# EPICS substitutions: blenApp/Db/lcls2/blen_gap_coefI2.substitutions
#======================================
# Register with DoubleVal interfaces
#======================================

file "RegisterDoubleOut.template" { pattern
{ P,              R,            DESC,                   PINI,  SCAN,        PORT,        EGU,          PARAM      }
{ $(P),     $(AMC):CoefI2,        "Coef I2 - Offset",            "YES",  "Passive",   $(PORT),     "",     AMC$(AMC):CoefI2  }
}

file "RegisterDoubleOutRBV.template" { pattern
{ P,              R,            DESC,                   PINI,  SCAN,        PORT,        EGU,          PARAM      }
{ $(P),     $(AMC):CoefI2RBV,     "Coef I2- Offset",            "YES", "1 second",  $(PORT),     "",     AMC$(AMC):CoefI2  }
}
